// TwinCAT 3 PLC project HT_Standard
// Title: HT_Standard
// Company: Help-tec Automation AG
// Author: Roger Schluep
// ProjectVersion: 0.3.0
// Description: Help-tec standard library
// ProgramVersion: 3.1.4023.0
// libraries:
//   Tc2_Standard, * (Beckhoff Automation GmbH)
//   Tc3_Module, * (Beckhoff Automation GmbH)
//   TcUnit, * (www.tcunit.org)
// project tree:
//   Cylinder/ CylinderMonostable.TcPOU, CylinderBistable.TcPOU, CylinderTimingConfig.TcDUT, eCylinderError.TcDUT, eCylinderStep.TcDUT, Simu_CylinderBistable.TcPOU, Simu_CylinderMonostable.TcPOU
//   HMI/ ButtonHMI.TcPOU, ButtonLongPress.TcPOU, ButtonTrig.TcPOU, ButtonPress.TcPOU
//   / PlcTask.TcTTO
//   Test/ ButtonPress_Test.TcPOU, ButtonTrig_Test.TcPOU, CylinderMonostable_Test.TcPOU, CylinderBistable_Test.TcPOU, PRG_TEST.TcPOU
// real-time tasks:
//   TASK PlcTask: cycle T#10ms, priority 20, ADS port 350

CONFIGURATION HT_Standard
    RESOURCE PLC ON TwinCAT3
        TASK PlcTask(INTERVAL := T#10ms, PRIORITY := 20);
        PROGRAM PRG_TEST WITH PlcTask : PRG_TEST;
    END_RESOURCE
END_CONFIGURATION

// ---- Cylinder/CylinderTimingConfig.TcDUT
/// timing configuration for FINAL standard cylinder 2 positions
TYPE CylinderTimingConfig :
STRUCT
    alarmToHomePos_time : TIME := T#3S; // maximum allowed travel time from work pos to home pos sensor
    alarmToWorkPos_time : TIME := T#3S; // maximum allowed travel time from home pos to work pos sensor

    atHomePos_time : TIME := T#100MS; // extra waiting time before considaring the cylinder to be in home pos
    atWorkPos_time : TIME := T#100MS; // extra waiting time before considaring the cylinder to be in work pos

    sensorFilterTime : TIME := T#250MS; // Filter the possible flickering of sensor
END_STRUCT
END_TYPE

// ---- Cylinder/eCylinderError.TcDUT
{attribute 'qualified_only'}
{attribute 'to_string'}
TYPE eCylinderError :
(
    none                           := 0,
    sensorHomeAndWorkBothActivated := 1,
    sensorInHomePosDisapeared      := 2,
    timeoutMoveInWorkPos           := 3,
    sensorInWorkPosDisapeared      := 4,
    timeoutMoveInHomePos           := 5,
    inErrorState                   := 6,
    uknownStepNumber               := 7,

    _max
) UDINT;
END_TYPE

// ---- Cylinder/eCylinderStep.TcDUT
{attribute 'qualified_only'}
{attribute 'strict'}
TYPE INTERNAL eCylinderStep :
(
    RESET,
    IN_HOME_POS,
    MOVE_TO_WORK_POS,
    IN_WORK_POS,
    MOVE_TO_HOME_POS,
    ERROR
);
END_TYPE

// ---- Test/PRG_TEST.TcPOU
PROGRAM INTERNAL PRG_TEST
VAR
    _buttonPress_Test        : ButtonPress_Test;
    _buttonTrig_Test         : ButtonTrig_Test;
    _cylinderMonostable_Test : CylinderMonostable_Test;
    _cylinderBistable_Test   : CylinderBistable_Test;
END_VAR

TcUnit.RUN();

END_PROGRAM

// ---- Test/ButtonPress_Test.TcPOU
FUNCTION_BLOCK INTERNAL ButtonPress_Test EXTENDS TcUnit.FB_TestSuite
VAR_INPUT
END_VAR
VAR_OUTPUT
END_VAR
VAR
END_VAR

outputsTestsWithAllInputFalse();

hmiSignalOutputTest();

buttonDisableTest();

METHOD buttonDisableTest
VAR_INPUT
END_VAR
VAR
    bp : ButtonPress;
END_VAR
TEST('buttonDisableTest');

// init fb
bp.inDisable := FALSE;
bp.inOn      := FALSE;
bp.inError   := FALSE;
bp();

(********** TEST 1 **********)

// Simulate a HMI press signal
bp.SetButton(TRUE);

// first call
bp(inDisable := TRUE);

AssertEquals_BOOL(Expected := FALSE,
                  Actual   := bp.outPress,
                  Message  := 'ButtonPress must be FALSE when desactivated');

// second call
bp(inDisable := FALSE);

AssertEquals_BOOL(Expected := TRUE,
                  Actual   := bp.outPress,
                  Message  := 'ButtonPress must be TRUE when activated again');

TEST_FINISHED();
END_METHOD

METHOD hmiSignalOutputTest
VAR_INPUT
END_VAR
VAR
    bp : ButtonPress;
END_VAR
TEST('hmiSignalOutputTest');

(* TEST 1 *)
bp(inDisable := FALSE,
   inOn      := FALSE,
   inError   := FALSE);

AssertEquals_BOOL(Expected := FALSE,
                  Actual   := bp._disable,
                  Message  := 'TEST 1: button._disable is not FALSE');

AssertEquals_BOOL(Expected := FALSE,
                  Actual   := bp._on,
                  Message  := 'TEST 1: button._on is not FALSE');

AssertEquals_BOOL(Expected := FALSE,
                  Actual   := bp._error,
                  Message  := 'TEST 1: button._error is not FALSE');

(* TEST 2 *)
bp(inDisable := TRUE,
   inOn      := FALSE,
   inError   := FALSE);

AssertEquals_BOOL(Expected := TRUE,
                  Actual   := bp._disable,
                  Message  := 'TEST 2: button._disable is not TRUE');

AssertEquals_BOOL(Expected := FALSE,
                  Actual   := bp._on,
                  Message  := 'TEST 2: button._on is not FALSE');

AssertEquals_BOOL(Expected := FALSE,
                  Actual   := bp._error,
                  Message  := 'TEST 2: button._error is not FALSE');

(* TEST 3 *)
bp(inDisable := TRUE,
   inOn      := TRUE,
   inError   := FALSE);

AssertEquals_BOOL(Expected := TRUE,
                  Actual   := bp._disable,
                  Message  := 'TEST 3: button._disable is not TRUE');

AssertEquals_BOOL(Expected := TRUE,
                  Actual   := bp._on,
                  Message  := 'TEST 3: button._on is not TRUE');

AssertEquals_BOOL(Expected := FALSE,
                  Actual   := bp._error,
                  Message  := 'TEST 3: button._error is not FALSE');

(* TEST 4 *)
bp(inDisable := TRUE,
   inOn      := TRUE,
   inError   := TRUE);

AssertEquals_BOOL(Expected := TRUE,
                  Actual   := bp._disable,
                  Message  := 'TEST 4: button._disable is not TRUE');

AssertEquals_BOOL(Expected := FALSE,
                  Actual   := bp._on,
                  Message  := 'TEST 4: button._on needs to be FALSE when inError is TRUE');

AssertEquals_BOOL(Expected := TRUE,
                  Actual   := bp._error,
                  Message  := 'TEST 4: button._error is not TRUE');

(* TEST 5 *)
bp(inDisable := FALSE,
   inOn      := FALSE,
   inError   := TRUE);

AssertEquals_BOOL(Expected := FALSE,
                  Actual   := bp._disable,
                  Message  := 'TEST 5: button._disable is not FALSE');

AssertEquals_BOOL(Expected := FALSE,
                  Actual   := bp._on,
                  Message  := 'TEST 5: button._on needs to be false when inError is TRUE');

AssertEquals_BOOL(Expected := TRUE,
                  Actual   := bp._error,
                  Message  := 'TEST 5: button._error is not TRUE');

TcUnit.TEST_FINISHED();
END_METHOD

METHOD outputsTestsWithAllInputFalse
VAR_INPUT
END_VAR
VAR
    bp : ButtonPress;
END_VAR
TEST('outputsTestsWithAllInputFalse');

// init fb
bp.inDisable := FALSE;
bp.inError   := FALSE;
bp.inOn      := FALSE;
bp();

(********** TEST 1 **********)

// Simulate a HMI press signal
bp.SetButton(TRUE);

// first call
bp();

AssertEquals_BOOL(Expected := TRUE,
                  Actual   := bp.outPress,
                  Message  := 'TEST 1: ButtonPress.outPress is not TRUE');

AssertEquals_BOOL(Expected := TRUE,
                  Actual   := bp.outRisingEdge,
                  Message  := 'TEST 1: ButtonPress.outRisingEdge is not TRUE');

AssertEquals_BOOL(Expected := FALSE,
                  Actual   := bp.outFallingEdge,
                  Message  := 'TEST 1: ButtonPress.outFallingEdge is not FALSE');

(********** TEST 2 **********)
// second call
bp();

AssertEquals_BOOL(Expected := TRUE,
                  Actual   := bp.outPress,
                  Message  := 'TEST 2: ButtonPress.outPress must be TRUE');

AssertEquals_BOOL(Expected := FALSE,
                  Actual   := bp.outRisingEdge,
                  Message  := 'TEST 2: ButtonPress.outRisingEdge is not FALSE');

AssertEquals_BOOL(Expected := FALSE,
                  Actual   := bp.outFallingEdge,
                  Message  := 'TEST 2: ButtonPress.outFallingEdge is not FALSE');

(********** TEST 3 **********)

// release button from HMI
bp.SetButton(FALSE);

// first call (with new input value)
bp();

AssertEquals_BOOL(Expected := FALSE,
                  Actual   := bp.outPress,
                  Message  := 'TEST 3: ButtonPress.outPress is not FALSE');

AssertEquals_BOOL(Expected := FALSE,
                  Actual   := bp.outRisingEdge,
                  Message  := 'TEST 3: ButtonPress.outRisingEdge is not FALSE');

AssertEquals_BOOL(Expected := TRUE,
                  Actual   := bp.outFallingEdge,
                  Message  := 'TEST 3: ButtonPress.outFallingEdge is not TRUE');

(********** TEST 4 **********)

// second call (with button as false)
bp();

AssertEquals_BOOL(Expected := FALSE,
                  Actual   := bp.outPress,
                  Message  := 'TEST 4: ButtonPress.outPress is not FALSE');

AssertEquals_BOOL(Expected := FALSE,
                  Actual   := bp.outRisingEdge,
                  Message  := 'TEST 4: ButtonPress.outRisingEdge is not FALSE');

AssertEquals_BOOL(Expected := FALSE,
                  Actual   := bp.outFallingEdge,
                  Message  := 'TEST 4: ButtonPress.outFallingEdge is not FALSE');

TEST_FINISHED();
END_METHOD

END_FUNCTION_BLOCK

// ---- HMI/ButtonPress.TcPOU
FUNCTION_BLOCK PUBLIC ButtonPress EXTENDS ButtonHMI
VAR_INPUT
END_VAR
VAR_OUTPUT
    outPress       : BOOL;
    outRisingEdge  : BOOL;
    outFallingEdge : BOOL;
END_VAR
VAR
    _clk : BOOL; // used to generate the R_Trig and F_Trig
END_VAR

_disable := inDisable;
_on      := inOn AND NOT inError;
_error   := inError;

outPress       := _button AND NOT inDisable;
outRisingEdge  := _button AND NOT _clk AND NOT inDisable;
outFallingEdge := NOT _button AND _clk AND NOT inDisable;

_clk := _button;

END_FUNCTION_BLOCK

// ---- HMI/ButtonHMI.TcPOU
FUNCTION_BLOCK ABSTRACT ButtonHMI
VAR_INPUT
    inDisable : BOOL; // disable the button and show the 'disable' state of the button
    inOn      : BOOL; // show the 'on' state of the button
    inError   : BOOL; // show the 'error' state of the button
END_VAR
VAR_OUTPUT
END_VAR
VAR
    _button  : BOOL; // link this variable to the output of your HMI button
    _disable : BOOL; // link this variable to the 'disable' input of your HMI button
    _on      : BOOL; // link this variable to the 'on' input of your HMI button
    _error   : BOOL; // link this variable to the 'error' or 'alarm' input of your HMI button
END_VAR

/// Set the internal button state
/// used to bypass the HMI action
METHOD PUBLIC SetButton
VAR_INPUT
    value : BOOL;
END_VAR
THIS^._button := value;
END_METHOD

END_FUNCTION_BLOCK

// ---- Test/ButtonTrig_Test.TcPOU
FUNCTION_BLOCK INTERNAL ButtonTrig_Test EXTENDS ButtonPress_Test
VAR_INPUT
END_VAR
VAR_OUTPUT
END_VAR
VAR
END_VAR

outputsTestsWithAllInputFalse();

hmiSignalOutputTest();

buttonDisableTest();

LongPressTest();

METHOD buttonDisableTest
VAR_INPUT
END_VAR
VAR
    bp : ButtonTrig;
END_VAR
TEST('buttonDisableTest');

// init fb
bp.inDisable := FALSE;
bp.inOn      := FALSE;
bp.inError   := FALSE;
bp();

(********** TEST 1 **********)

// Simulate a HMI press signal
bp.SetButton(TRUE);

// first call
bp(inDisable := TRUE);

AssertEquals_BOOL(Expected := FALSE,
                  Actual   := bp.outRisingEdge,
                  Message  := 'ButtonTrig must be FALSE when desactivated');

// second call
bp(inDisable := FALSE);

AssertEquals_BOOL(Expected := FALSE,
                  Actual   := bp.outRisingEdge,
                  Message  := 'ButtonTrig must stay false even after disable signal is released');

TEST_FINISHED();
END_METHOD

METHOD hmiSignalOutputTest
VAR_INPUT
END_VAR
VAR
    bp : ButtonTrig;
END_VAR
TEST('hmiSignalOutputTest');

(* TEST 1 *)
bp(inDisable := FALSE,
   inOn      := FALSE,
   inError   := FALSE);

AssertEquals_BOOL(Expected := FALSE,
                  Actual   := bp._disable,
                  Message  := 'TEST 1: ButtonTrig._disable is not FALSE');

AssertEquals_BOOL(Expected := FALSE,
                  Actual   := bp._on,
                  Message  := 'TEST 1: ButtonTrig._on is not FALSE');

AssertEquals_BOOL(Expected := FALSE,
                  Actual   := bp._error,
                  Message  := 'TEST 1: ButtonTrig._error is not FALSE');

(* TEST 2 *)
bp(inDisable := TRUE,
   inOn      := FALSE,
   inError   := FALSE);

AssertEquals_BOOL(Expected := TRUE,
                  Actual   := bp._disable,
                  Message  := 'TEST 2: ButtonTrig._disable is not TRUE');

AssertEquals_BOOL(Expected := FALSE,
                  Actual   := bp._on,
                  Message  := 'TEST 2: ButtonTrig._on is not FALSE');

AssertEquals_BOOL(Expected := FALSE,
                  Actual   := bp._error,
                  Message  := 'TEST 2: ButtonTrig._error is not FALSE');

(* TEST 3 *)
bp(inDisable := TRUE,
   inOn      := TRUE,
   inError   := FALSE);

AssertEquals_BOOL(Expected := TRUE,
                  Actual   := bp._disable,
                  Message  := 'TEST 3: ButtonTrig._disable is not TRUE');

AssertEquals_BOOL(Expected := TRUE,
                  Actual   := bp._on,
                  Message  := 'TEST 3: ButtonTrig._on is not TRUE');

AssertEquals_BOOL(Expected := FALSE,
                  Actual   := bp._error,
                  Message  := 'TEST 3: ButtonTrig._error is not FALSE');

(* TEST 4 *)
bp(inDisable := TRUE,
   inOn      := TRUE,
   inError   := TRUE);

AssertEquals_BOOL(Expected := TRUE,
                  Actual   := bp._disable,
                  Message  := 'TEST 4: ButtonTrig._disable is not TRUE');

AssertEquals_BOOL(Expected := FALSE,
                  Actual   := bp._on,
                  Message  := 'TEST 4: ButtonTrig._on needs to be FALSE when inError is TRUE');

AssertEquals_BOOL(Expected := TRUE,
                  Actual   := bp._error,
                  Message  := 'TEST 4: ButtonTrig._error is not TRUE');

(* TEST 5 *)
bp(inDisable := FALSE,
   inOn      := FALSE,
   inError   := TRUE);

AssertEquals_BOOL(Expected := FALSE,
                  Actual   := bp._disable,
                  Message  := 'TEST 5: ButtonTrig._disable is not FALSE');

AssertEquals_BOOL(Expected := FALSE,
                  Actual   := bp._on,
                  Message  := 'TEST 5: ButtonTrig._on needs to be false when inError is TRUE');

AssertEquals_BOOL(Expected := TRUE,
                  Actual   := bp._error,
                  Message  := 'TEST 5: ButtonTrig._error is not TRUE');

TcUnit.TEST_FINISHED();
END_METHOD

METHOD LongPressTest
VAR_INPUT
END_VAR
VAR
    bp : ButtonTrig;
END_VAR
TEST('LongPressTest for ButtonTrig');

(* TEST 1 *)
bp(inDisable := FALSE,
   inOn      := FALSE,
   inError   := FALSE);

bp.SetButton(TRUE);
bp();

AssertTrue(bp.outRisingEdge, 'At the first call, bp.outRisingEdge must be TRUE');

// stay pressed with the HMI
bp.SetButton(TRUE);
bp();

AssertFalse(bp.outRisingEdge,
            'At the second call, bp.outRisingEdge must be FALSE even if the HMI force the button to be on');

bp.SetButton(FALSE);
bp();

AssertFalse(bp.outRisingEdge, 'outRisingEdge must be FALSE');

bp.SetButton(TRUE);
bp();

AssertTrue(bp.outRisingEdge, 'outRisingEdge must be TRUE right after the rising edge of _button');

TcUnit.TEST_FINISHED();
END_METHOD

METHOD outputsTestsWithAllInputFalse
VAR_INPUT
END_VAR
VAR
    bp : ButtonTrig;
END_VAR
TEST('outputsTestsWithAllInputFalse');

// init fb
bp.inDisable := FALSE;
bp.inError   := FALSE;
bp.inOn      := FALSE;
bp();

(********** TEST 1 **********)

// Simulate a HMI press signal
bp.SetButton(TRUE);

// first call
bp();

AssertEquals_BOOL(Expected := TRUE,
                  Actual   := bp.outRisingEdge,
                  Message  := 'TEST 1: ButtonPress.outRisingEdge is not TRUE');

(********** TEST 2 **********)
// second call
bp();

AssertEquals_BOOL(Expected := FALSE,
                  Actual   := bp.outRisingEdge,
                  Message  := 'TEST 2: ButtonPress.outRisingEdge is not FALSE');

(********** TEST 3 **********)

// release button from HMI
bp.SetButton(FALSE);

// first call (with new input value)
bp();

AssertEquals_BOOL(Expected := FALSE,
                  Actual   := bp.outRisingEdge,
                  Message  := 'TEST 3: ButtonPress.outRisingEdge is not FALSE');

(********** TEST 4 **********)

// second call (with new input value)
bp();

AssertEquals_BOOL(Expected := FALSE,
                  Actual   := bp.outRisingEdge,
                  Message  := 'TEST 4: ButtonPress.outRisingEdge is not FALSE');

TEST_FINISHED();
END_METHOD

END_FUNCTION_BLOCK

// ---- HMI/ButtonTrig.TcPOU
FUNCTION_BLOCK PUBLIC ButtonTrig EXTENDS ButtonHMI
VAR_INPUT
END_VAR
VAR_OUTPUT
    outRisingEdge : BOOL;
END_VAR
VAR
    _clk : BOOL; // used to generate the R_Trig
END_VAR

_disable := inDisable;
_on      := inOn AND NOT inError;
_error   := inError;

outRisingEdge := _button AND NOT _clk AND NOT inDisable;

_clk := _button;

_button := FALSE;

END_FUNCTION_BLOCK

// ---- Test/CylinderMonostable_Test.TcPOU
FUNCTION_BLOCK INTERNAL CylinderMonostable_Test EXTENDS FB_TestSuite
VAR_INPUT
END_VAR
VAR_OUTPUT
END_VAR
VAR
    _cylinder     : CylinderMonostable;
    _timingConfig : CylinderTimingConfig := (alarmToHomePos_time := T#1S,
                                             alarmToWorkPos_time := T#1S,
                                             atHomePos_time := T#100MS,
                                             atWorkPos_time := T#100MS,
                                             SensorFilterTime := T#250MS);

    _travelTime : TIME := T#200MS;

END_VAR

THIS^.InitCylinder(_cylinder, 'testWithoutError');
THIS^.OpenCylinder(_cylinder, 'open test');
THIS^.CloseCylinder(_cylinder);
THIS^.ErrorWhileOpening(_cylinder);
THIS^.ErrorAck(_cylinder, 'ack error opening');
THIS^.ErrorWhileClosing(_cylinder);
THIS^.ErrorAck(_cylinder, 'ack error closing');
THIS^.CloseCylinderDuringOpening(_cylinder);
THIS^.OpenCylinder(_cylinder, 'open for HomeCylinderDuringWork test');
THIS^.HomeCylinderDuringWork(_cylinder);

METHOD CloseCylinder
VAR_INPUT
    refCylinder : REFERENCE TO CylinderMonostable;
END_VAR
VAR_INST
    simulateTravel_ton : Tc2_Standard.TON;
    timeout_ton        : Tc2_Standard.TON;
END_VAR

IF TcUnit.TEST_ORDERED('CloseCylinder') THEN

    refCylinder(inGoToPosHome      := TRUE,
                inGoToPosWork      := FALSE,
                inAtPosHome_sensor := simulateTravel_ton.Q,
                inAtPosWork_sensor := refCylinder.outAtPosWork);

    simulateTravel_ton(IN := refCylinder.inGoToPosHome, PT := THIS^._travelTime);
    timeout_ton(IN := refCylinder.inAtPosHome_sensor, PT := THIS^._timingConfig.atHomePos_time);

    IF refCylinder.outAtPosHome THEN
        AssertTrue(refCylinder.outAtPosHome, 'outInHomePos is not TRUE');
        AssertFalse(refCylinder.outAtPosWork, 'outInWorkPos is not FASE');

        simulateTravel_ton(IN := FALSE);
        timeout_ton(IN := FALSE);
        TcUnit.TEST_FINISHED();

    ELSIF timeout_ton.Q THEN
        AssertTrue(FALSE, 'Cylinder not in home pos in time');
        simulateTravel_ton(IN := FALSE);
        timeout_ton(IN := FALSE);
        TcUnit.TEST_FINISHED();
    END_IF

END_IF
END_METHOD

METHOD CloseCylinderDuringOpening
VAR_INPUT
    refCylinder : REFERENCE TO CylinderMonostable;
END_VAR
VAR_INST
    simulateOpening_ton       : Tc2_Standard.TON; // Use to open the cylinder a bit before closing it again
    simulateClosingTravel_ton : Tc2_Standard.TON;
    timeout_ton               : Tc2_Standard.TON;
END_VAR
VAR CONSTANT
    TEST_CYLINDER_OPENING_PHASE_NAME : STRING := 'CloseCylinderDuringOpening - opening phase';
    TEST_CYLINDER_CLOSING_PHASE_NAME : STRING := 'CloseCylinderDuringOpening - closing phase';
END_VAR

IF TcUnit.TEST_ORDERED(TEST_CYLINDER_OPENING_PHASE_NAME) THEN

    refCylinder(inGoToPosHome      := FALSE,
                inGoToPosWork      := TRUE,
                inAtPosHome_sensor := refCylinder.outAtPosHome,
                inAtPosWork_sensor := FALSE);

    simulateOpening_ton(IN := refCylinder.inGoToPosWork, PT := THIS^._travelTime / 2);

    IF simulateOpening_ton.Q THEN
        AssertFalse(refCylinder.outAtPosHome, 'outInHomePos is not FASE');
        AssertFalse(refCylinder.outAtPosWork, 'outInWorkPos is not FASE');

        TcUnit.TEST_FINISHED_NAMED(TEST_CYLINDER_OPENING_PHASE_NAME);
    END_IF

END_IF

IF TcUnit.TEST_ORDERED(TEST_CYLINDER_CLOSING_PHASE_NAME) THEN

    refCylinder(inGoToPosHome      := TRUE,
                inGoToPosWork      := FALSE,
                inAtPosHome_sensor := simulateClosingTravel_ton.Q,
                inAtPosWork_sensor := FALSE);

    simulateClosingTravel_ton(IN := NOT refCylinder.outValvePosWork, PT := THIS^._travelTime / 2);
    timeout_ton(IN := refCylinder.inAtPosHome_sensor, PT := THIS^._timingConfig.atHomePos_time);

    AssertFalse(refCylinder.outAtPosWork, 'cylinder must not reach its work position in this situation');
    AssertFalse(refCylinder.outValvePosWork, 'outValveWorkPos must turned off when we move in home again');

    IF refCylinder.outAtPosHome THEN
        AssertTrue(refCylinder.outAtPosHome, 'outInHomePos is not TRUE');
        AssertFalse(refCylinder.outAtPosWork, 'outInWorkPos is not FASE');

        TcUnit.TEST_FINISHED_NAMED(TEST_CYLINDER_CLOSING_PHASE_NAME);

    ELSIF timeout_ton.Q THEN
        AssertTrue(FALSE, 'Cylinder not in home pos in time');
        TcUnit.TEST_FINISHED_NAMED(TEST_CYLINDER_CLOSING_PHASE_NAME);

    ELSIF refCylinder.outError THEN
        AssertTrue(FALSE, 'Cylinder in error - timeout of the command. Other test may failed due to this error');
        TcUnit.TEST_FINISHED_NAMED(TEST_CYLINDER_CLOSING_PHASE_NAME);
    END_IF
END_IF
END_METHOD

METHOD ErrorAck
VAR_INPUT
    refCylinder : REFERENCE TO CylinderMonostable;
    testName    : STRING;
END_VAR
VAR
    errorAckCylinderTest_name : STRING := Tc2_Standard.CONCAT('Error Ack ', testName);
END_VAR
VAR_INST
END_VAR
IF TcUnit.TEST_ORDERED(errorAckCylinderTest_name) THEN

    refCylinder(inErrorAck := TRUE);

    AssertFalse(refCylinder.outAtPosHome, 'outInHomePos is not FALSE');
    AssertFalse(refCylinder.outAtPosWork, 'outInWorkPos is not FALSE');
    AssertFalse(refCylinder.outError, 'outError is not FALSE');
    AssertEquals_UDINT(refCylinder.outErrorID, 0, 'Error ID do not match');

    TcUnit.TEST_FINISHED_NAMED(errorAckCylinderTest_name);

END_IF
END_METHOD

METHOD ErrorWhileClosing
VAR_INPUT
    refCylinder : REFERENCE TO CylinderMonostable;
END_VAR
VAR
    errorCylinderTest_name : STRING := 'ErrorWhileClosing';
END_VAR
VAR_INST
    travelTime_ton : Tc2_Standard.TON;
END_VAR
IF TcUnit.TEST_ORDERED(errorCylinderTest_name) THEN

    refCylinder(inGoToPosHome      := TRUE,
                inGoToPosWork      := FALSE,
                inAtPosHome_sensor := FALSE,
                inAtPosWork_sensor := refCylinder.outAtPosWork);

    travelTime_ton(IN := TRUE, PT := THIS^._timingConfig.alarmToHomePos_time);

    IF travelTime_ton.Q THEN
        AssertFalse(refCylinder.outAtPosHome, 'outInHomePos is not FALSE');
        AssertFalse(refCylinder.outAtPosWork, 'outInWorkPos is not FALSE');
        AssertTrue(refCylinder.outError, 'outError is not TRUE');
        AssertEquals_UDINT(refCylinder.outErrorID,
                           eCylinderError.timeoutMoveInHomePos,
                           'Error ID do not match');

        travelTime_ton(IN := FALSE);

        // set the sensor to prevent further error
        _cylinder(inAtPosHome_sensor := TRUE);

        TcUnit.TEST_FINISHED_NAMED(errorCylinderTest_name);
    END_IF

END_IF
END_METHOD

METHOD ErrorWhileOpening
VAR_INPUT
    refCylinder : REFERENCE TO CylinderMonostable;
END_VAR
VAR
    errorCylinderTest_name : STRING := 'ErrorWhileOpening';
END_VAR
VAR_INST
    travelTime_ton : Tc2_Standard.TON;
END_VAR
IF TcUnit.TEST_ORDERED(errorCylinderTest_name) THEN

    refCylinder(inGoToPosHome      := FALSE,
                inGoToPosWork      := TRUE,
                inAtPosHome_sensor := refCylinder.outAtPosHome,
                inAtPosWork_sensor := FALSE);

    travelTime_ton(IN := TRUE, PT := THIS^._timingConfig.alarmToWorkPos_time);

    IF travelTime_ton.Q THEN
        AssertFalse(refCylinder.outAtPosHome, 'outInHomePos is not FALSE');
        AssertFalse(refCylinder.outAtPosWork, 'outInWorkPos is not FALSE');
        AssertTrue(refCylinder.outError, 'outError is not TRUE');
        AssertEquals_UDINT(refCylinder.outErrorID,
                           eCylinderError.timeoutMoveInWorkPos,
                           'Error ID do not match');

        travelTime_ton(IN := FALSE);

        // set the sensor to prevent further error
        _cylinder(inAtPosWork_sensor := TRUE);

        TcUnit.TEST_FINISHED_NAMED(errorCylinderTest_name);
    END_IF

END_IF
END_METHOD

METHOD HomeCylinderDuringWork
VAR_INPUT
    refCylinder : REFERENCE TO CylinderMonostable;
END_VAR
VAR_INST
    simulateClosing_ton       : Tc2_Standard.TON; // Use to close the cylinder a bit before closing it again
    simulateOpeningTravel_ton : Tc2_Standard.TON;
    timeout_ton               : Tc2_Standard.TON;
END_VAR
VAR CONSTANT
    TEST_CYLINDER_CLOSING_PHASE_NAME : STRING := 'HomeCylinderDuringWork - closing phase';
    TEST_CYLINDER_OPENING_PHASE_NAME : STRING := 'HomeCylinderDuringWork - opening phase';
END_VAR

IF TcUnit.TEST_ORDERED(TEST_CYLINDER_CLOSING_PHASE_NAME) THEN

    refCylinder(inGoToPosHome      := TRUE,
                inGoToPosWork      := FALSE,
                inAtPosHome_sensor := FALSE,
                inAtPosWork_sensor := refCylinder.outAtPosWork);

    simulateClosing_ton(IN := refCylinder.inGoToPosHome, PT := THIS^._travelTime / 2);

    IF simulateClosing_ton.Q THEN
        AssertFalse(refCylinder.outAtPosHome, 'outInHomePos is not FASE');
        AssertFalse(refCylinder.outAtPosWork, 'outInWorkPos is not FASE');

        TcUnit.TEST_FINISHED_NAMED(TEST_CYLINDER_CLOSING_PHASE_NAME);
    END_IF

END_IF

IF TcUnit.TEST_ORDERED(TEST_CYLINDER_OPENING_PHASE_NAME) THEN

    refCylinder(inGoToPosHome      := FALSE,
                inGoToPosWork      := TRUE,
                inAtPosHome_sensor := FALSE,
                inAtPosWork_sensor := simulateOpeningTravel_ton.Q);

    simulateOpeningTravel_ton(IN := refCylinder.outValvePosWork, PT := THIS^._travelTime / 2);
    timeout_ton(IN := refCylinder.inAtPosWork_sensor, PT := THIS^._timingConfig.atWorkPos_time);

    AssertFalse(refCylinder.outAtPosHome, 'cylinder must not reach its home position in this situation');
    AssertTrue(refCylinder.outValvePosWork, 'outValveWorkPos must be on when we move in work again');

    IF refCylinder.outAtPosWork THEN
        AssertFalse(refCylinder.outAtPosHome, 'outInHomePos is not FALSE');
        AssertTrue(refCylinder.outAtPosWork, 'outInWorkPos is not TRUE');

        TcUnit.TEST_FINISHED_NAMED(TEST_CYLINDER_OPENING_PHASE_NAME);

    ELSIF timeout_ton.Q THEN
        AssertTrue(FALSE, 'Cylinder not in home pos in time');
        TcUnit.TEST_FINISHED_NAMED(TEST_CYLINDER_OPENING_PHASE_NAME);

    ELSIF refCylinder.outError THEN
        AssertTrue(FALSE, 'Cylinder in error - timeout of the command. Other test may failed due to this error');
        TcUnit.TEST_FINISHED_NAMED(TEST_CYLINDER_OPENING_PHASE_NAME);
    END_IF
END_IF
END_METHOD

METHOD InitCylinder
VAR_INPUT
    refCylinder    : REFERENCE TO CylinderMonostable;
    initTestDefine : STRING;
END_VAR
VAR
    testInitCylinder_name : STRING := Tc2_Standard.CONCAT('InitCylinder-', initTestDefine);
    testHomeCylinder_name : STRING := Tc2_Standard.CONCAT('Wait cylinder to be in home pos-', initTestDefine);
END_VAR
VAR_INST
    simulateTravel_ton : Tc2_Standard.TON;
END_VAR

IF TcUnit.TEST_ORDERED(testInitCylinder_name) THEN

    refCylinder(inReset            := FALSE,
                inErrorAck         := FALSE,
                inManualMode       := FALSE,
                inGoToPosHome      := FALSE,
                inGoToPosWork      := FALSE,
                inAtPosHome_sensor := FALSE,
                inAtPosWork_sensor := FALSE,
                inTimingConfig     := THIS^._timingConfig);

    AssertFalse(refCylinder.outValvePosWork, 'default position must be at home pos');
    AssertFalse(refCylinder.outAtPosHome, 'at the begining the cylinder must not be at home pos, yet');
    AssertFalse(refCylinder.outAtPosWork, 'outInWorkPos is not FALSE');
    AssertFalse(refCylinder.outError, 'outError is not FALSE');
    AssertFalse(refCylinder.outErrorID <> 0, 'outErrorID must be 0 if there is no error');

    TcUnit.TEST_FINISHED_NAMED(testInitCylinder_name);
END_IF

IF TcUnit.TEST_ORDERED(testHomeCylinder_name) THEN

    refCylinder(inAtPosHome_sensor := TRUE,
                inAtPosWork_sensor := FALSE);

    simulateTravel_ton(IN := refCylinder.inAtPosHome_sensor, PT := THIS^._timingConfig.atHomePos_time);

    IF simulateTravel_ton.Q THEN
        AssertFalse(refCylinder.outValvePosWork, 'outValveWorkPos is not FALSE');
        AssertTrue(refCylinder.outAtPosHome, 'outInHomePos must be TRUE');
        AssertFalse(refCylinder.outAtPosWork, 'outInWorkPos is not FALSE');
        AssertFalse(refCylinder.outError, 'outError is not FALSE');
        AssertFalse(refCylinder.outErrorID <> 0, 'outErrorID must be 0 if there is no error');

        TcUnit.TEST_FINISHED_NAMED(testHomeCylinder_name);
    END_IF
END_IF
END_METHOD

METHOD OpenCylinder
VAR_INPUT
    refCylinder : REFERENCE TO CylinderMonostable;
    testName    : STRING;
END_VAR
VAR
    openCylinderTest_name : STRING := Tc2_Standard.CONCAT('OpenCylinder', testName);
END_VAR
VAR_INST
    simulateTravel_ton : Tc2_Standard.TON;
    timeout_ton        : Tc2_Standard.TON;
END_VAR

IF TcUnit.TEST_ORDERED(openCylinderTest_name) THEN

    refCylinder(inGoToPosHome      := FALSE,
                inGoToPosWork      := TRUE,
                inAtPosHome_sensor := refCylinder.outAtPosHome,
                inAtPosWork_sensor := simulateTravel_ton.Q);

    simulateTravel_ton(IN := refCylinder.inGoToPosWork, PT := THIS^._travelTime);
    timeout_ton(IN := refCylinder.inAtPosWork_sensor, PT := THIS^._timingConfig.atWorkPos_time);

    IF refCylinder.outAtPosWork THEN
        AssertFalse(refCylinder.outAtPosHome, 'outInHomePos is not FALSE');

        AssertTrue(refCylinder.outAtPosWork, 'outInWorkPos is not TRUE');

        simulateTravel_ton(IN := FALSE);
        timeout_ton(IN := FALSE);
        TcUnit.TEST_FINISHED();

    ELSIF timeout_ton.Q THEN
        AssertTRUE(FALSE, 'Cylinder not in work pos in time');
        simulateTravel_ton(IN := FALSE);
        timeout_ton(IN := FALSE);
        TcUnit.TEST_FINISHED();
    END_IF

END_IF
END_METHOD

END_FUNCTION_BLOCK

// ---- Cylinder/CylinderMonostable.TcPOU
/// Manage a monostable valve
/// use inGoToHomePos and inGoToWorkPos to command the valve
/// inGoToHomePos has precedence to inGoToWorkPos
FUNCTION_BLOCK PUBLIC CylinderMonostable
VAR_INPUT
    inReset      : BOOL; // Force the valve to stay in place
    inErrorAck   : BOOL;
    inManualMode : BOOL;

    inGoToPosHome : BOOL;
    inGoToPosWork : BOOL;

    inAtPosHome_sensor : BOOL; // feedback sensor to confirm home position
    inAtPosWork_sensor : BOOL; // feedback sensor to confirm work position

    inTimingConfig : CylinderTimingConfig;

END_VAR
VAR_OUTPUT
    outValvePosWork : BOOL;
    outAtPosHome    : BOOL;
    outAtPosWork    : BOOL;
    outError        : BOOL;
    outErrorID      : UDINT;
    outErrorString  : STRING;
END_VAR
VAR
    _state            : eCylinderStep;
    _stateBeforeError : eCylinderStep;

    _bpManu : ButtonTrig;

    TON_ErrAS             : Tc2_Standard.TON;
    TON_ErrGS             : Tc2_Standard.TON;
    TOF_sensorHomePosLost : Tc2_Standard.TOF;
    TOF_sensorWorkPosLost : Tc2_Standard.TOF;
    TON_GS_AS             : Tc2_Standard.TON;
    TON_WaitAS            : Tc2_Standard.TON;
    TON_WaitGS            : Tc2_Standard.TON;
END_VAR

// inGoToWorkPos can not be TRUE if inGoToHomePos is TRUE
inGoToPosWork := inGoToPosWork AND NOT inGoToPosHome;

IF inReset THEN
    _stateBeforeError := eCylinderStep.RESET;
    _state            := eCylinderStep.RESET;
END_IF

IF inErrorAck AND (outErrorID <> 0) THEN
    outErrorID := 0;
    _state     := _stateBeforeError;
END_IF

_bpManu(inDisable := NOT inManualMode,
        inOn      := outAtPosWork,
        inError   := outError);

// We update the timer to notice an error
TON_ErrGS();

// We update the timer to notice an error
TON_ErrAS();

TOF_sensorHomePosLost(IN := inAtPosHome_sensor,
                      PT := inTimingConfig.sensorFilterTime);

TOF_sensorWorkPosLost(IN := inAtPosWork_sensor,
                      PT := inTimingConfig.sensorFilterTime);

TON_GS_AS(IN := inAtPosHome_sensor AND inAtPosWork_sensor,
          PT := inTimingConfig.sensorFilterTime);

TON_WaitGS(in := inAtPosHome_sensor,
           PT := inTimingConfig.atHomePos_time);

TON_WaitAS(in := inAtPosWork_sensor,
           PT := inTimingConfig.atWorkPos_time);

IF TON_GS_AS.Q THEN
    outErrorID        := eCylinderError.sensorHomeAndWorkBothActivated;
    _stateBeforeError := eCylinderStep.RESET;
    _state            := eCylinderStep.ERROR;
END_IF

CASE _state OF

eCylinderStep.RESET:
    IF NOT inReset THEN
        IF inAtPosHome_sensor THEN
            _state := eCylinderStep.IN_HOME_POS;
        ELSIF inAtPosWork_sensor THEN
            _state := eCylinderStep.IN_WORK_POS;
        ELSIF outValvePosWork THEN
            _state := eCylinderStep.MOVE_TO_WORK_POS;
        ELSE
            _state := eCylinderStep.MOVE_TO_HOME_POS;
        END_IF
    END_IF

eCylinderStep.IN_HOME_POS:
    IF inManualMode THEN
        IF _bpManu.outRisingEdge THEN
            _state := eCylinderStep.MOVE_TO_WORK_POS;
        END_IF
    ELSIF inGoToPosWork THEN
        _state := eCylinderStep.MOVE_TO_WORK_POS;
    ELSIF NOT TOF_sensorHomePosLost.Q THEN
        outErrorID        := eCylinderError.sensorInHomePosDisapeared;
        _stateBeforeError := eCylinderStep.MOVE_TO_HOME_POS;
        _state            := eCylinderStep.ERROR;
    END_IF

eCylinderStep.MOVE_TO_WORK_POS:
    IF TON_WaitAS.Q OR inManualMode THEN
        _state := eCylinderStep.IN_WORK_POS;
    ELSIF inGoToPosHome THEN
        _state := eCylinderStep.MOVE_TO_HOME_POS;
    ELSIF TON_ErrAS.Q THEN
        outErrorID        := eCylinderError.timeoutMoveInWorkPos;
        _stateBeforeError := eCylinderStep.MOVE_TO_WORK_POS;
        _state            := eCylinderStep.ERROR;
    END_IF

eCylinderStep.IN_WORK_POS:
    IF inManualMode THEN
        IF _bpManu.outRisingEdge THEN
            _state := eCylinderStep.MOVE_TO_HOME_POS;
        END_IF
    ELSIF inGoToPosHome THEN
        _state := eCylinderStep.MOVE_TO_HOME_POS;
    ELSIF NOT TOF_sensorWorkPosLost.Q THEN
        outErrorID        := eCylinderError.sensorInWorkPosDisapeared;
        _stateBeforeError := eCylinderStep.MOVE_TO_WORK_POS;
        _state            := eCylinderStep.ERROR;
    END_IF

eCylinderStep.MOVE_TO_HOME_POS:
    IF TON_WaitGS.Q OR inManualMode THEN
        _state := eCylinderStep.IN_HOME_POS;
    ELSIF inGoToPosWork THEN
        _state := eCylinderStep.MOVE_TO_WORK_POS;
    ELSIF TON_ErrGS.Q THEN
        outErrorID        := eCylinderError.timeoutMoveInHomePos;
        _stateBeforeError := eCylinderStep.MOVE_TO_HOME_POS;
        _state            := eCylinderStep.ERROR;
    END_IF

eCylinderStep.ERROR:
    IF (outErrorID = 0) THEN
        outErrorID := eCylinderError.inErrorState;
    END_IF;

ELSE
    outErrorID := eCylinderError.uknownStepNumber;
    _state     := eCylinderStep.ERROR;
END_CASE

IF (_state <> eCylinderStep.RESET) AND (_state <> eCylinderStep.ERROR) THEN
    outValvePosWork := (_state = eCylinderStep.MOVE_TO_WORK_POS) OR (_state = eCylinderStep.IN_WORK_POS);
END_IF

// We have to update the timer here to be able to match the timing error
TON_ErrGS(in := (_state = eCylinderStep.MOVE_TO_HOME_POS) AND NOT inAtPosHome_sensor,
          pt := inTimingConfig.alarmToHomePos_time);

// We have to update the timer here to be able to match the timing error
TON_ErrAS(in := (_state = eCylinderStep.MOVE_TO_WORK_POS) AND NOT inAtPosWork_sensor,
          pt := inTimingConfig.alarmToWorkPos_time);

outAtPosHome   := (_state = eCylinderStep.IN_HOME_POS);
outAtPosWork   := (_state = eCylinderStep.IN_WORK_POS);
outError       := (outErrorID <> 0);
outErrorID     := outErrorID;
outErrorString := TO_STRING(outErrorID);

END_FUNCTION_BLOCK

// ---- Test/CylinderBistable_Test.TcPOU
FUNCTION_BLOCK INTERNAL CylinderBistable_Test EXTENDS FB_TestSuite
VAR_INPUT
END_VAR
VAR_OUTPUT
END_VAR
VAR
    _cylinder     : CylinderBistable;
    _timingConfig : CylinderTimingConfig := (alarmToHomePos_time := T#1S,
                                             alarmToWorkPos_time := T#1S,
                                             atHomePos_time := T#100MS,
                                             atWorkPos_time := T#100MS,
                                             SensorFilterTime := T#250MS);

    _travelTime : TIME := T#200MS;

END_VAR

THIS^.InitCylinder(_cylinder, 'testWithoutError');
THIS^.OpenCylinder(_cylinder, 'open test');
THIS^.CloseCylinder(_cylinder);
THIS^.ErrorWhileOpening(_cylinder);
THIS^.ErrorAck(_cylinder, 'ack error opening');
THIS^.ErrorWhileClosing(_cylinder);
THIS^.ErrorAck(_cylinder, 'ack error closing');
THIS^.CloseCylinderDuringOpening(_cylinder);
THIS^.OpenCylinder(_cylinder, 'open for HomeCylinderDuringWork test');
THIS^.HomeCylinderDuringWork(_cylinder);

METHOD CloseCylinder
VAR_INPUT
    refCylinder : REFERENCE TO CylinderMonostable;
END_VAR
VAR_INST
    simulateTravel_ton : Tc2_Standard.TON;
    timeout_ton        : Tc2_Standard.TON;
END_VAR

IF TcUnit.TEST_ORDERED('CloseCylinder') THEN

    refCylinder(inGoToPosHome      := TRUE,
                inGoToPosWork      := FALSE,
                inAtPosHome_sensor := simulateTravel_ton.Q,
                inAtPosWork_sensor := refCylinder.outAtPosWork);

    simulateTravel_ton(IN := refCylinder.inGoToPosHome, PT := THIS^._travelTime);
    timeout_ton(IN := refCylinder.inAtPosHome_sensor, PT := THIS^._timingConfig.atHomePos_time);

    IF refCylinder.outAtPosHome THEN
        AssertTrue(refCylinder.outAtPosHome, 'outInHomePos is not TRUE');
        AssertFalse(refCylinder.outAtPosWork, 'outInWorkPos is not FASE');

        simulateTravel_ton(IN := FALSE);
        timeout_ton(IN := FALSE);
        TcUnit.TEST_FINISHED();

    ELSIF timeout_ton.Q THEN
        AssertTrue(FALSE, 'Cylinder not in home pos in time');
        simulateTravel_ton(IN := FALSE);
        timeout_ton(IN := FALSE);
        TcUnit.TEST_FINISHED();
    END_IF

END_IF
END_METHOD

METHOD CloseCylinderDuringOpening
VAR_INPUT
    refCylinder : REFERENCE TO CylinderBistable;
END_VAR
VAR_INST
    simulateOpening_ton       : Tc2_Standard.TON; // Use to open the cylinder a bit before closing it again
    simulateClosingTravel_ton : Tc2_Standard.TON;
    timeout_ton               : Tc2_Standard.TON;
END_VAR
VAR CONSTANT
    TEST_CYLINDER_OPENING_PHASE_NAME : STRING := 'CloseCylinderDuringOpening - opening phase';
    TEST_CYLINDER_CLOSING_PHASE_NAME : STRING := 'CloseCylinderDuringOpening - closing phase';
END_VAR

IF TcUnit.TEST_ORDERED(TEST_CYLINDER_OPENING_PHASE_NAME) THEN

    refCylinder(inGoToPosHome      := FALSE,
                inGoToPosWork      := TRUE,
                inAtPosHome_sensor := refCylinder.outAtPosHome,
                inAtPosWork_sensor := FALSE);

    simulateOpening_ton(IN := refCylinder.inGoToPosWork, PT := THIS^._travelTime / 2);

    IF simulateOpening_ton.Q THEN
        AssertFalse(refCylinder.outAtPosHome, 'outInHomePos is not FASE');
        AssertFalse(refCylinder.outAtPosWork, 'outInWorkPos is not FASE');

        TcUnit.TEST_FINISHED_NAMED(TEST_CYLINDER_OPENING_PHASE_NAME);
    END_IF

END_IF

IF TcUnit.TEST_ORDERED(TEST_CYLINDER_CLOSING_PHASE_NAME) THEN

    refCylinder(inGoToPosHome      := TRUE,
                inGoToPosWork      := FALSE,
                inAtPosHome_sensor := simulateClosingTravel_ton.Q,
                inAtPosWork_sensor := FALSE);

    simulateClosingTravel_ton(IN := refCylinder.outValvePosHome, PT := THIS^._travelTime / 2);
    timeout_ton(IN := refCylinder.inAtPosHome_sensor, PT := THIS^._timingConfig.atHomePos_time);

    AssertFalse(refCylinder.outAtPosWork, 'cylinder must not reach its work position in this situation');
    AssertFalse(refCylinder.outValvePosWork, 'outValveWorkPos must turned off when we move in home again');

    IF refCylinder.outAtPosHome THEN
        AssertTrue(refCylinder.outAtPosHome, 'outInHomePos is not TRUE');
        AssertFalse(refCylinder.outAtPosWork, 'outInWorkPos is not FASE');

        TcUnit.TEST_FINISHED_NAMED(TEST_CYLINDER_CLOSING_PHASE_NAME);

    ELSIF timeout_ton.Q THEN
        AssertTrue(FALSE, 'Cylinder not in home pos in time');
        TcUnit.TEST_FINISHED_NAMED(TEST_CYLINDER_CLOSING_PHASE_NAME);

    ELSIF refCylinder.outError THEN
        AssertTrue(FALSE, 'Cylinder in error - timeout of the command. Other test may failed due to this error');
        TcUnit.TEST_FINISHED_NAMED(TEST_CYLINDER_CLOSING_PHASE_NAME);
    END_IF
END_IF
END_METHOD

METHOD ErrorAck
VAR_INPUT
    refCylinder : REFERENCE TO CylinderMonostable;
    testName    : STRING;
END_VAR
VAR
    errorAckCylinderTest_name : STRING := Tc2_Standard.CONCAT('Error Ack ', testName);
END_VAR
VAR_INST
END_VAR
IF TcUnit.TEST_ORDERED(errorAckCylinderTest_name) THEN

    refCylinder(inErrorAck := TRUE);

    AssertFalse(refCylinder.outAtPosHome, 'outInHomePos is not FALSE');
    AssertFalse(refCylinder.outAtPosWork, 'outInWorkPos is not FALSE');
    AssertFalse(refCylinder.outError, 'outError is not FALSE');
    AssertEquals_UDINT(refCylinder.outErrorID, 0, 'Error ID do not match');

    TcUnit.TEST_FINISHED_NAMED(errorAckCylinderTest_name);

END_IF
END_METHOD

METHOD ErrorWhileClosing
VAR_INPUT
    refCylinder : REFERENCE TO CylinderMonostable;
END_VAR
VAR
    errorCylinderTest_name : STRING := 'ErrorWhileClosing';
END_VAR
VAR_INST
    travelTime_ton : Tc2_Standard.TON;
END_VAR
IF TcUnit.TEST_ORDERED(errorCylinderTest_name) THEN

    refCylinder(inGoToPosHome      := TRUE,
                inGoToPosWork      := FALSE,
                inAtPosHome_sensor := FALSE,
                inAtPosWork_sensor := refCylinder.outAtPosWork);

    travelTime_ton(IN := TRUE, PT := THIS^._timingConfig.alarmToHomePos_time);

    IF travelTime_ton.Q THEN
        AssertFalse(refCylinder.outAtPosHome, 'outInHomePos is not FALSE');
        AssertFalse(refCylinder.outAtPosWork, 'outInWorkPos is not FALSE');
        AssertTrue(refCylinder.outError, 'outError is not TRUE');
        AssertEquals_UDINT(refCylinder.outErrorID,
                           eCylinderError.timeoutMoveInHomePos,
                           'Error ID do not match');

        travelTime_ton(IN := FALSE);

        // set the sensor to prevent further error
        _cylinder(inAtPosHome_sensor := TRUE);

        TcUnit.TEST_FINISHED_NAMED(errorCylinderTest_name);
    END_IF

END_IF
END_METHOD

METHOD ErrorWhileOpening
VAR_INPUT
    refCylinder : REFERENCE TO CylinderMonostable;
END_VAR
VAR
    errorCylinderTest_name : STRING := 'ErrorWhileOpening';
END_VAR
VAR_INST
    travelTime_ton : Tc2_Standard.TON;
END_VAR
IF TcUnit.TEST_ORDERED(errorCylinderTest_name) THEN

    refCylinder(inGoToPosHome      := FALSE,
                inGoToPosWork      := TRUE,
                inAtPosHome_sensor := refCylinder.outAtPosHome,
                inAtPosWork_sensor := FALSE);

    travelTime_ton(IN := TRUE, PT := THIS^._timingConfig.alarmToWorkPos_time);

    IF travelTime_ton.Q THEN
        AssertFalse(refCylinder.outAtPosHome, 'outInHomePos is not FALSE');
        AssertFalse(refCylinder.outAtPosWork, 'outInWorkPos is not FALSE');
        AssertTrue(refCylinder.outError, 'outError is not TRUE');
        AssertEquals_UDINT(refCylinder.outErrorID,
                           eCylinderError.timeoutMoveInWorkPos,
                           'Error ID do not match');

        travelTime_ton(IN := FALSE);

        // set the sensor to prevent further error
        _cylinder(inAtPosWork_sensor := TRUE);

        TcUnit.TEST_FINISHED_NAMED(errorCylinderTest_name);
    END_IF

END_IF
END_METHOD

METHOD HomeCylinderDuringWork
VAR_INPUT
    refCylinder : REFERENCE TO CylinderBistable;
END_VAR
VAR_INST
    simulateClosing_ton       : Tc2_Standard.TON; // Use to close the cylinder a bit before closing it again
    simulateOpeningTravel_ton : Tc2_Standard.TON;
    timeout_ton               : Tc2_Standard.TON;
END_VAR
VAR CONSTANT
    TEST_CYLINDER_CLOSING_PHASE_NAME : STRING := 'HomeCylinderDuringWork - closing phase';
    TEST_CYLINDER_OPENING_PHASE_NAME : STRING := 'HomeCylinderDuringWork - opening phase';
END_VAR

IF TcUnit.TEST_ORDERED(TEST_CYLINDER_CLOSING_PHASE_NAME) THEN

    refCylinder(inGoToPosHome      := TRUE,
                inGoToPosWork      := FALSE,
                inAtPosHome_sensor := FALSE,
                inAtPosWork_sensor := refCylinder.outAtPosWork);

    simulateClosing_ton(IN := refCylinder.inGoToPosHome, PT := THIS^._travelTime / 2);

    IF simulateClosing_ton.Q THEN
        AssertFalse(refCylinder.outAtPosHome, 'outInHomePos is not FASE');
        AssertFalse(refCylinder.outAtPosWork, 'outInWorkPos is not FASE');

        TcUnit.TEST_FINISHED_NAMED(TEST_CYLINDER_CLOSING_PHASE_NAME);
    END_IF

END_IF

IF TcUnit.TEST_ORDERED(TEST_CYLINDER_OPENING_PHASE_NAME) THEN

    refCylinder(inGoToPosHome      := FALSE,
                inGoToPosWork      := TRUE,
                inAtPosHome_sensor := FALSE,
                inAtPosWork_sensor := simulateOpeningTravel_ton.Q);

    simulateOpeningTravel_ton(IN := refCylinder.outValvePosWork, PT := THIS^._travelTime / 2);
    timeout_ton(IN := refCylinder.inAtPosWork_sensor, PT := THIS^._timingConfig.atWorkPos_time);

    AssertFalse(refCylinder.outAtPosHome, 'cylinder must not reach its home position in this situation');
    AssertFalse(refCylinder.outValvePosHome, 'outValvePosHome must not be on when we move in work again');

    IF refCylinder.outAtPosWork THEN
        AssertFalse(refCylinder.outAtPosHome, 'outInHomePos is not FALSE');
        AssertTrue(refCylinder.outAtPosWork, 'outInWorkPos is not TRUE');

        TcUnit.TEST_FINISHED_NAMED(TEST_CYLINDER_OPENING_PHASE_NAME);

    ELSIF timeout_ton.Q THEN
        AssertTrue(FALSE, 'Cylinder not in home pos in time');
        TcUnit.TEST_FINISHED_NAMED(TEST_CYLINDER_OPENING_PHASE_NAME);

    ELSIF refCylinder.outError THEN
        AssertTrue(FALSE, 'Cylinder in error - timeout of the command. Other test may failed due to this error');
        TcUnit.TEST_FINISHED_NAMED(TEST_CYLINDER_OPENING_PHASE_NAME);
    END_IF
END_IF
END_METHOD

METHOD InitCylinder
VAR_INPUT
    refCylinder    : REFERENCE TO CylinderMonostable;
    initTestDefine : STRING;
END_VAR
VAR
    testInitCylinder_name : STRING := Tc2_Standard.CONCAT('InitCylinder-', initTestDefine);
    testHomeCylinder_name : STRING := Tc2_Standard.CONCAT('Wait cylinder to be in home pos-', initTestDefine);
END_VAR
VAR_INST
    simulateTravel_ton : Tc2_Standard.TON;
END_VAR

IF TcUnit.TEST_ORDERED(testInitCylinder_name) THEN

    refCylinder(inReset            := FALSE,
                inErrorAck         := FALSE,
                inManualMode       := FALSE,
                inGoToPosHome      := FALSE,
                inGoToPosWork      := FALSE,
                inAtPosHome_sensor := FALSE,
                inAtPosWork_sensor := FALSE,
                inTimingConfig     := THIS^._timingConfig);

    AssertFalse(refCylinder.outValvePosWork, 'default position must be at home pos');
    AssertFalse(refCylinder.outAtPosHome, 'at the begining the cylinder must not be at home pos, yet');
    AssertFalse(refCylinder.outAtPosWork, 'outInWorkPos is not FALSE');
    AssertFalse(refCylinder.outError, 'outError is not FALSE');
    AssertFalse(refCylinder.outErrorID <> 0, 'outErrorID must be 0 if there is no error');

    TcUnit.TEST_FINISHED_NAMED(testInitCylinder_name);
END_IF

IF TcUnit.TEST_ORDERED(testHomeCylinder_name) THEN

    refCylinder(inAtPosHome_sensor := TRUE,
                inAtPosWork_sensor := FALSE);

    simulateTravel_ton(IN := refCylinder.inAtPosHome_sensor, PT := THIS^._timingConfig.atHomePos_time);

    IF simulateTravel_ton.Q THEN
        AssertFalse(refCylinder.outValvePosWork, 'outValveWorkPos is not FALSE');
        AssertTrue(refCylinder.outAtPosHome, 'outInHomePos must be TRUE');
        AssertFalse(refCylinder.outAtPosWork, 'outInWorkPos is not FALSE');
        AssertFalse(refCylinder.outError, 'outError is not FALSE');
        AssertFalse(refCylinder.outErrorID <> 0, 'outErrorID must be 0 if there is no error');

        TcUnit.TEST_FINISHED_NAMED(testHomeCylinder_name);
    END_IF
END_IF
END_METHOD

METHOD OpenCylinder
VAR_INPUT
    refCylinder : REFERENCE TO CylinderMonostable;
    testName    : STRING;
END_VAR
VAR
    openCylinderTest_name : STRING := Tc2_Standard.CONCAT('OpenCylinder', testName);
END_VAR
VAR_INST
    simulateTravel_ton : Tc2_Standard.TON;
    timeout_ton        : Tc2_Standard.TON;
END_VAR

IF TcUnit.TEST_ORDERED(openCylinderTest_name) THEN

    refCylinder(inGoToPosHome      := FALSE,
                inGoToPosWork      := TRUE,
                inAtPosHome_sensor := refCylinder.outAtPosHome,
                inAtPosWork_sensor := simulateTravel_ton.Q);

    simulateTravel_ton(IN := refCylinder.inGoToPosWork, PT := THIS^._travelTime);
    timeout_ton(IN := refCylinder.inAtPosWork_sensor, PT := THIS^._timingConfig.atWorkPos_time);

    IF refCylinder.outAtPosWork THEN
        AssertFalse(refCylinder.outAtPosHome, 'outInHomePos is not FALSE');

        AssertTrue(refCylinder.outAtPosWork, 'outInWorkPos is not TRUE');

        simulateTravel_ton(IN := FALSE);
        timeout_ton(IN := FALSE);
        TcUnit.TEST_FINISHED();

    ELSIF timeout_ton.Q THEN
        AssertTRUE(FALSE, 'Cylinder not in work pos in time');
        simulateTravel_ton(IN := FALSE);
        timeout_ton(IN := FALSE);
        TcUnit.TEST_FINISHED();
    END_IF

END_IF
END_METHOD

END_FUNCTION_BLOCK

// ---- Cylinder/CylinderBistable.TcPOU
/// Manage a bistable valve
/// use inGoToHomePos and inGoToWorkPos to command the valve
/// inGoToHomePos has precedence to inGoToWorkPos
/// This FB only activate the corresponding output of the
/// valve during the travel of the cylinder
FUNCTION_BLOCK PUBLIC CylinderBistable EXTENDS CylinderMonostable
VAR_OUTPUT
    outValvePosHome : BOOL;
END_VAR

SUPER^();

IF (_state <> eCylinderStep.RESET) AND (_state <> eCylinderStep.ERROR) THEN
    outValvePosHome := (_state = eCylinderStep.MOVE_TO_HOME_POS);
    // @Override
    outValvePosWork := (_state = eCylinderStep.MOVE_TO_WORK_POS);
END_IF

END_FUNCTION_BLOCK

// ---- Cylinder/Simu_CylinderBistable.TcPOU
/// Simulate a cylinder movement.
/// Work with CylinderBistable
FUNCTION_BLOCK Simu_CylinderBistable
VAR_INPUT
    inEnable                : BOOL; // enable the simulation of a the connected Cylinder
    inRefCylinder           : REFERENCE TO CylinderBistable;
    inAtPosHome_sensor      : BOOL;
    inAtPosWork_sensor      : BOOL;
    inToHomePositionTime_ms : DINT; // time in ms when GS signal should be on
    inToWorkPositionTime_ms : DINT; // time in ms when AS signal should be on
END_VAR
VAR
    ton_ToHomePosition : Tc2_Standard.TON;
    ton_ToWorkPosition : Tc2_Standard.TON;
END_VAR


IF NOT __ISVALIDREF(inRefCylinder) THEN
    RETURN;
END_IF

ton_ToHomePosition(IN := inRefCylinder.outValvePosHome OR
                         (inRefCylinder._state = eCylinderStep.IN_HOME_POS),
                   PT := DINT_TO_TIME(inToHomePositionTime_ms));

ton_ToWorkPosition(IN := inRefCylinder.outValvePosWork OR
                         (inRefCylinder._state = eCylinderStep.IN_WORK_POS),
                   PT := DINT_TO_TIME(inToWorkPositionTime_ms));

inRefCylinder.inAtPosHome_sensor := (inEnable AND ton_ToHomePosition.Q) OR
                                    (NOT inEnable AND inAtPosHome_sensor);

inRefCylinder.inAtPosWork_sensor := (inEnable AND ton_ToWorkPosition.Q) OR
                                    (NOT inEnable AND inAtPosWork_sensor);

END_FUNCTION_BLOCK

// ---- Cylinder/Simu_CylinderMonostable.TcPOU
/// Simulate a cylinder movement.
/// Work with CylinderMonostable
FUNCTION_BLOCK Simu_CylinderMonostable
VAR_INPUT
    inEnable                : BOOL; // enable the simulation of a the connected Cylinder
    inRefCylinder           : REFERENCE TO CylinderMonostable;
    inAtPosHome_sensor      : BOOL;
    inAtPosWork_sensor      : BOOL;
    inToHomePositionTime_ms : DINT; // time in ms when GS signal should be on
    inToWorkPositionTime_ms : DINT; // time in ms when AS signal should be on
END_VAR
VAR
    ton_ToHomePosition : Tc2_Standard.TON;
    ton_ToWorkPosition : Tc2_Standard.TON;
END_VAR


IF NOT __ISVALIDREF(inRefCylinder) THEN
    RETURN;
END_IF

ton_ToHomePosition(IN := NOT inRefCylinder.outValvePosWork,
                   PT := DINT_TO_TIME(inToHomePositionTime_ms));

ton_ToWorkPosition(IN := inRefCylinder.outValvePosWork,
                   PT := DINT_TO_TIME(inToWorkPositionTime_ms));

inRefCylinder.inAtPosHome_sensor := (inEnable AND ton_ToHomePosition.Q) OR
                                    (NOT inEnable AND inAtPosHome_sensor);

inRefCylinder.inAtPosWork_sensor := (inEnable AND ton_ToWorkPosition.Q) OR
                                    (NOT inEnable AND inAtPosWork_sensor);

END_FUNCTION_BLOCK

// ---- HMI/ButtonLongPress.TcPOU
// The button must be pressed for a given time
// to activate its outputs
FUNCTION_BLOCK ButtonLongPress EXTENDS ButtonPress
VAR_INPUT
    inPressTime : TIME;
END_VAR
VAR_OUTPUT
END_VAR
VAR
    _tonPressTime : Tc2_Standard.TON;
END_VAR

_tonPressTime(IN := _button AND NOT inDisable,
              PT := inPressTime);

_disable := inDisable;
_on      := inOn AND NOT inError;
_error   := inError;

outPress       := _tonPressTime.Q AND NOT inDisable;
outRisingEdge  := _tonPressTime.Q AND NOT _clk AND NOT inDisable;
outFallingEdge := NOT _tonPressTime.Q AND _clk AND NOT inDisable;

_clk := _tonPressTime.Q;

END_FUNCTION_BLOCK
